// TIA Portal V18 export
TYPE "UDT_WSsAI"
// stored: IsFailsafeCompliant false
   STRUCT
      r14200a : Real;   // 14.200a
      r14201a : Real;   // 14.201a
   END_STRUCT;
END_TYPE
